% RSLogix 500 project conveyor final.RSS, saved by version 8.30.00.16 %
PROJECT "UNTITLED"    % processor: Bul.1763 MicroLogix 1100 Series B %

PROGRAM FILES
  LAD 2   6 rungs

DATA FILES
  O0 OUTPUT  4 elements
  I1 INPUT  6 elements
  S2 STATUS  66 elements
  B3 BINARY  1 elements
  T4 TIMER  1 elements
  C5 COUNTER  1 elements
  R6 CONTROL  1 elements
  N7 INTEGER  1 elements
  F8 FLOAT  1 elements

LADDER 2
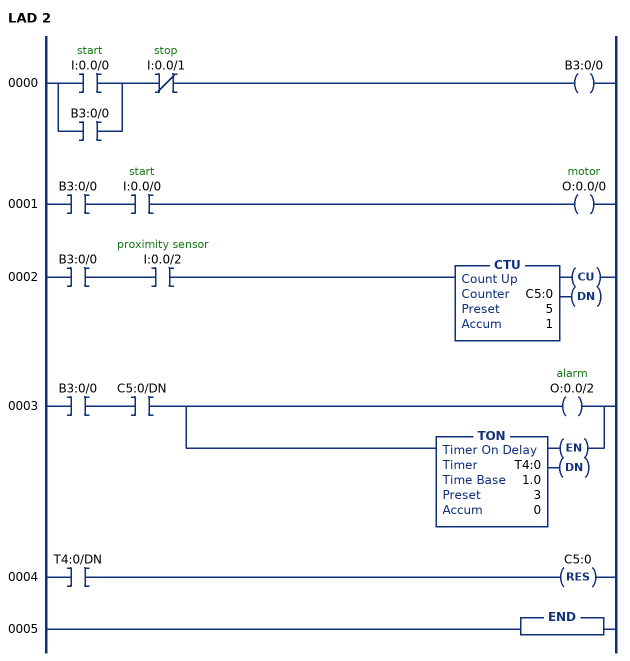
% Rung: 0 %
SOR BST XIC I:0.0/0 NXB XIC B3:0/0 BND XIO I:0.0/1 OTE B3:0/0 EOR
%   I:0.0/0  "start" %
%   I:0.0/1  "stop" %
% Rung: 1 %
SOR XIC B3:0/0 XIC I:0.0/0 OTE O:0.0/0 EOR
%   I:0.0/0  "start" %
%   O:0.0/0  "motor" %
% Rung: 2 %
SOR XIC B3:0/0 XIC I:0.0/2 CTU C5:0 5 1 EOR
%   I:0.0/2  "proximity sensor" %
% Rung: 3 %
SOR XIC B3:0/0 XIC C5:0/DN BST OTE O:0.0/2 NXB TON T4:0 1.0 3 0 BND EOR
%   O:0.0/2  "alarm" %
% Rung: 4 %
SOR XIC T4:0/DN RES C5:0 EOR
% Rung: 5 %
SOR END EOR

DATA TABLE (non-zero values as saved)
DATA B3
% B3:0 % 0X0001
DATA T4
% .PRE .ACC %
% T4:0 % 3 0
DATA C5
% .PRE .ACC %
% C5:0 % 5 1
